TYPE dut_Setting :
STRUCT
	Val: REAL;
	Desc: STRING;
	Unit: STRING;
	Minimum: REAL;
	Maximum: REAL;
	Write_level:REAL;
END_STRUCT
END_TYPE

(* stored: Version 1.1.0.1, ProductVersion 3.1.4024.0
   DUT dut_Setting: Id {ad366624-746e-4f94-9b8d-813fc1b5cb3c} *)
